// TIA Portal V20 export
TYPE "udt_Manual_Station"
   STRUCT
      Config : Struct
         TaktTime : Time;
         OperatorTaskTime : Time;
         FlowStepName : WString[10];
         NextStationFlowStepName : WString[10];
         StationNumber : Int;
         StationName : String[6];
         StationBypass : Bool;
         TAE_Enable : Bool;
         BlockedTimerPreset : Time;
      END_STRUCT;
      Takt : Struct
         RunTimer : Bool;
         ResetTimer : Bool;
         TimerPreset : Time;
         TimerValue : Time;
      END_STRUCT;
      OPMode : "OPMODE_OUT_UDT";
   END_STRUCT;
END_TYPE
